PROGRAM MacOperationTimeCtrl
VAR

END_VAR

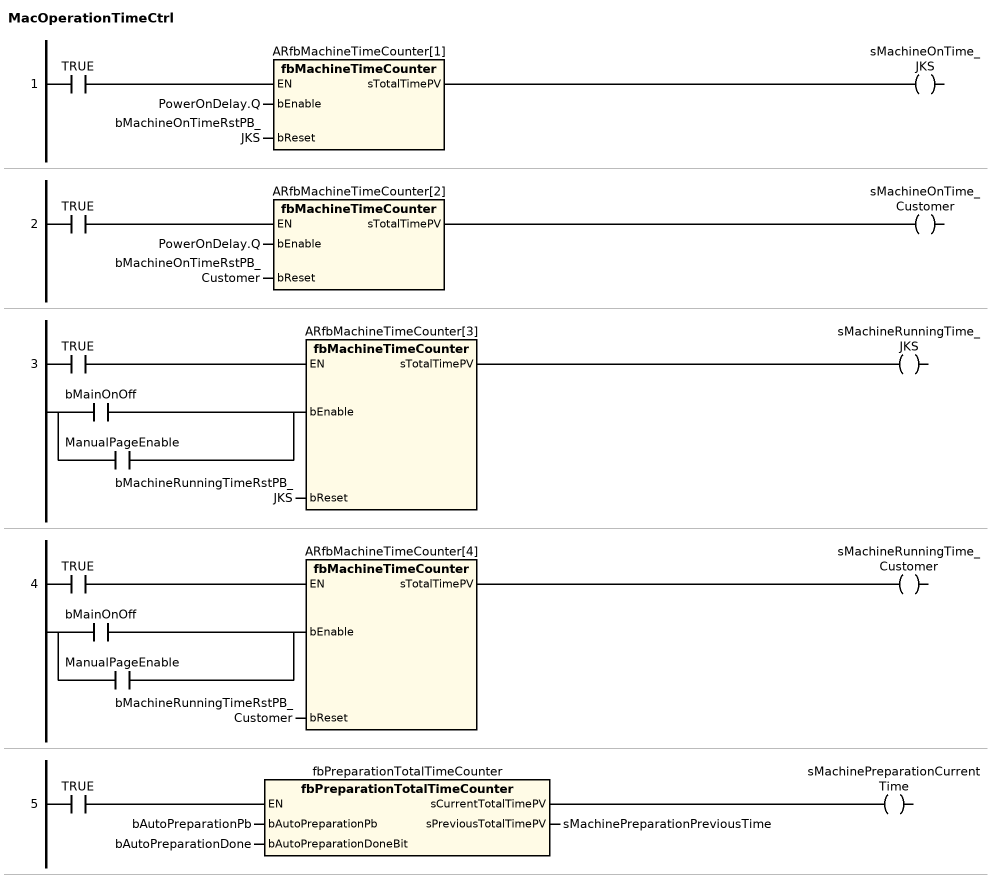
// NETWORK 1
ARfbMachineTimeCounter[1](bEnable := PowerOnDelay.Q, bReset := bMachineOnTimeRstPB_JKS); // fbMachineTimeCounter
sMachineOnTime_JKS := ARfbMachineTimeCounter[1].sTotalTimePV;

// NETWORK 2
ARfbMachineTimeCounter[2](bEnable := PowerOnDelay.Q, bReset := bMachineOnTimeRstPB_Customer); // fbMachineTimeCounter
sMachineOnTime_Customer := ARfbMachineTimeCounter[2].sTotalTimePV;

// NETWORK 3
ARfbMachineTimeCounter[3](bEnable := bMainOnOff OR ManualPageEnable, bReset := bMachineRunningTimeRstPB_JKS); // fbMachineTimeCounter
sMachineRunningTime_JKS := ARfbMachineTimeCounter[3].sTotalTimePV;

// NETWORK 4
ARfbMachineTimeCounter[4](bEnable := bMainOnOff OR ManualPageEnable, bReset := bMachineRunningTimeRstPB_Customer); // fbMachineTimeCounter
sMachineRunningTime_Customer := ARfbMachineTimeCounter[4].sTotalTimePV;

// NETWORK 5
fbPreparationTotalTimeCounter(
    bAutoPreparationPb := bAutoPreparationPb,
    bAutoPreparationDoneBit := bAutoPreparationDone,
    sPreviousTotalTimePV => sMachinePreparationPreviousTime);
sMachinePreparationCurrentTime := fbPreparationTotalTimeCounter.sCurrentTotalTimePV;

END_PROGRAM

(* stored: Version 1.1.0.1, ProductVersion 3.1.4024.12
   POU MacOperationTimeCtrl: Id {d2ba890b-27bf-4951-9f40-0734cdc71d69}, SpecialFunc None *)
